// TIA Portal V16 export
// export: Created 2022-09-01T13:36:48.4108243Z, ExportSetting WithDefaults, DisplayName Totally Integrated Automation Portal, DisplayVersion V16, DisplayName TIA Portal Version Control Interface, DisplayVersion V16, DisplayName TIA Portal Openness, DisplayVersion V16, DisplayName STEP 7 Professional, DisplayVersion V16, DisplayName STEP 7 Safety, DisplayVersion V16, DisplayName WinCC Advanced, DisplayVersion V16
FUNCTION "Proc_Analog_TK03" : Void   // FC9, LAD
{ S7_Optimized_Access := 'TRUE' }
VERSION : 0.1
// stored: AutoNumber true, IsIECCheckEnabled false, SetENOAutomatically false, UDAEnableTagReadback false
   VAR_INPUT
      Analog_Input_Value : Int;
   END_VAR
   VAR_OUTPUT
      Nível_em_metros : Real;
   END_VAR
   VAR_TEMP
      "Nível_em_%" : Real;
   END_VAR
BEGIN

REGION Network 1
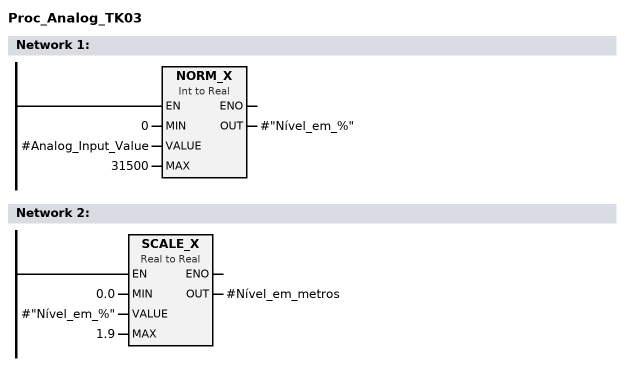
   RUNG wire#powerrail
      { S7_Templates := "[SrcType := Int, DestType := Real]"; S7_GenerateENO := "TRUE" } Normalize(min := 0, value := #Analog_Input_Value, max := 31500, out => #"Nível_em_%")
   END_RUNG
   // the same network as SCL:
   #"Nível_em_%" := NORM_X(MIN := 0, VALUE := #Analog_Input_Value, MAX := 31500);
END_REGION

REGION Network 2
   RUNG wire#powerrail
      { S7_Templates := "[SrcType := Real, DestType := Real]"; S7_GenerateENO := "TRUE" } Scale(min := 0.0, value := #"Nível_em_%", max := 1.9, out => #Nível_em_metros)
   END_RUNG
   // the same network as SCL:
   #Nível_em_metros := SCALE_X(MIN := 0.0, VALUE := #"Nível_em_%", MAX := 1.9);
END_REGION
END_FUNCTION
